// TwinCAT 3 PLC project Plc
// ProgramVersion: 3.1.4024.0
// libraries:
//   Tc2_Standard, * (Beckhoff Automation GmbH)
//   Tc2_System, * (Beckhoff Automation GmbH)
//   Tc3_Module, * (Beckhoff Automation GmbH)
//   VisuDialogs, * (System)
// project tree:
//   / Gestore di visualizzazione.TcVMO (not stored), GlobalTextList.TcGTLO, ImagePool.TcIPO (not stored), PlcTask.TcTTO (not stored), VisuTask.TcTTO
//   GVLs/ GVL.TcGVL
//   POUs/ MAIN.TcPOU, VISU.TcPOU (not stored)
//   VISUs/ Visualization.TcVIS
// real-time tasks:
//   TASK PlcTask: cycle T#10ms, priority 20, ADS port 350
//   TASK VisuTask: cycle T#100000us, priority 60, ADS port 351

CONFIGURATION Plc
    RESOURCE PLC ON TwinCAT3
        TASK VisuTask(INTERVAL := T#100000us, PRIORITY := 60);
        PROGRAM VISU WITH VisuTask : VISU;
    END_RESOURCE
END_CONFIGURATION

// ---- GVLs/GVL.TcGVL
{attribute 'qualified_only'}
VAR_GLOBAL
	//input
	PB1: BOOL; //Pulsante di start NA
	PB2: BOOL; //Pulsante di stop NC
	PBE: BOOL; //Pulsante di emergenza NC
	PS1: BOOL; //Fotocellula
	PS2: BOOL; //Fotocellula
	PS3: BOOL; //Fotocellula
	PS4: BOOL; //Fotocellula
	PS5: BOOL; //Fotocellula
	CS_BIANCO: BOOL; //Colore bianco rilevato
	CS_NERO: BOOL; //Colore nero rilevato
	
	//output
	L1: BOOL; //Luce di segnalazione bianca
	L2: BOOL; //Luce di segnalazione verde
	L3: BOOL; //Luce di segnalazione blue
	L4: BOOL; //Luce di segnalazione gialla
	L5: BOOL; //Luce di segnalazione rossa
	M1 : BOOL; //Motore nastro 1
	M2 : BOOL; //Motore nastro 2
	M3 : BOOL; //Motore discesa mandrino
	M4 : BOOL; //MOtore risalita mandrino
	M5 : BOOL; //Punta del trapano
	P1 : BOOL; //Pistone posizione intermedia
	P2 : BOOL; //Pistone posizione finale
	P3 : BOOL; //Pistone timbratura
	P4 : BOOL; //Pistone blocco pezzo
END_VAR

// ---- POUs/MAIN.TcPOU
PROGRAM MAIN
VAR
	//Stati
	IN_FUNZIONE: BOOL;
	IN_SMISTAMENTO: BOOL;
	IN_TIMBRATURA: BOOL;
	IN_FORATURA: BOOL;
	PEZZO_BIANCO: BOOL;
	PEZZO_NERO: BOOL;
	
	//Timer
	TON_BIANCO: TON;
	TON_NERO: TON;
	TON_TIMBRATURA: TON;
	TON_FORATURA_1: TON; // Il trapano scende in 2 secondi
	TON_FORATURA_2: TON; // Il trapano risale in 2 secondi

	//Counter
	CTU_BIANCHI: CTU;
	CTU_NERI: CTU;
	STOP_CONFERMATO: BOOL;
	STOP_RICHIESTO: BOOL;
	TON_STOP: TON;
	IN_ANOMALIA: BOOL;
	TON_ANOMALIA: TON;
	CONTROLLO_COLORE: BOOL;
	TON_ANOMALIA_COLORE: TON;
END_VAR

GestioneAnomalie();
GestioneStop();
GestionePulsantiSegnalazioni();
GestioneMotori();
GestioneSmistamento();
GestioneTimbratura();
GestioneForatura();
GestioneConteggio();

ACTION GestioneAnomalie:
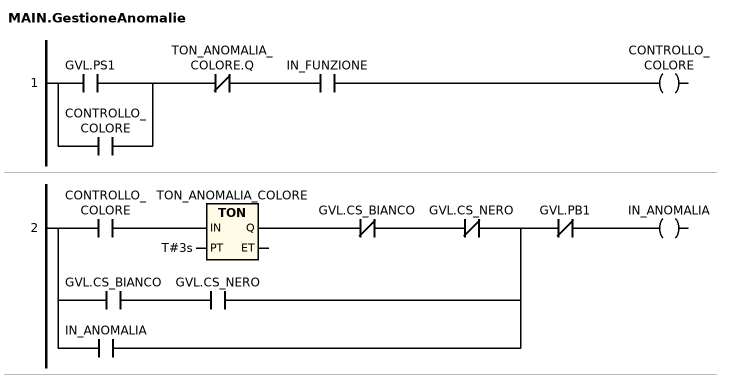
// NETWORK 1
CONTROLLO_COLORE := (GVL.PS1 OR CONTROLLO_COLORE) AND NOT TON_ANOMALIA_COLORE.Q AND IN_FUNZIONE;

// NETWORK 2
TON_ANOMALIA_COLORE(IN := CONTROLLO_COLORE, PT := T#3s); // TON
IN_ANOMALIA := (TON_ANOMALIA_COLORE.Q AND NOT GVL.CS_BIANCO AND NOT GVL.CS_NERO OR GVL.CS_BIANCO AND GVL.CS_NERO OR IN_ANOMALIA) AND NOT GVL.PB1;
END_ACTION

ACTION GestioneConteggio:
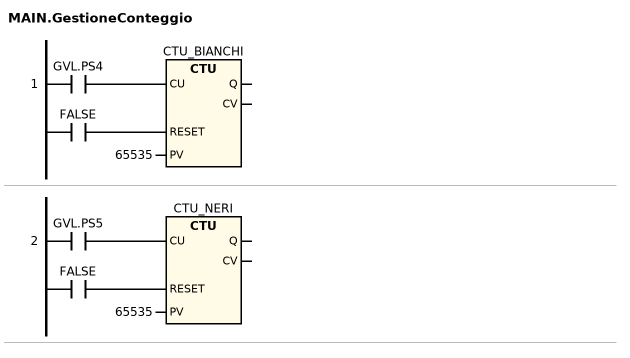
// NETWORK 1
CTU_BIANCHI(CU := GVL.PS4, RESET := FALSE, PV := 65535); // CTU

// NETWORK 2
CTU_NERI(CU := GVL.PS5, RESET := FALSE, PV := 65535); // CTU
END_ACTION

ACTION GestioneForatura:
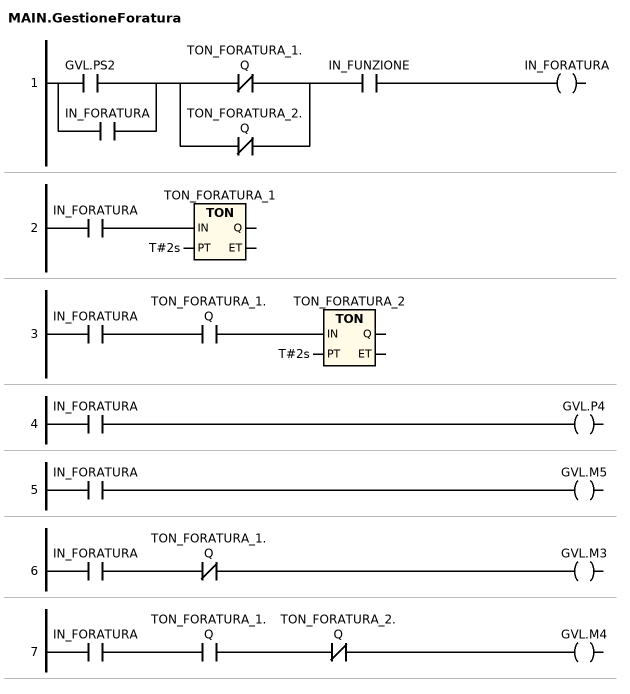
// NETWORK 1
IN_FORATURA := (GVL.PS2 OR IN_FORATURA) AND (NOT TON_FORATURA_1.Q OR NOT TON_FORATURA_2.Q) AND IN_FUNZIONE;

// NETWORK 2
TON_FORATURA_1(IN := IN_FORATURA, PT := T#2s); // TON

// NETWORK 3
TON_FORATURA_2(IN := IN_FORATURA AND TON_FORATURA_1.Q, PT := T#2s); // TON

// NETWORK 4
GVL.P4 := IN_FORATURA;

// NETWORK 5
GVL.M5 := IN_FORATURA;

// NETWORK 6
GVL.M3 := IN_FORATURA AND NOT TON_FORATURA_1.Q;

// NETWORK 7
GVL.M4 := IN_FORATURA AND TON_FORATURA_1.Q AND NOT TON_FORATURA_2.Q;
END_ACTION

ACTION GestioneMotori:
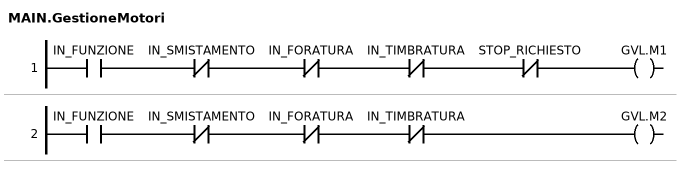
// NETWORK 1
GVL.M1 := IN_FUNZIONE AND NOT IN_SMISTAMENTO AND NOT IN_FORATURA AND NOT IN_TIMBRATURA AND NOT STOP_RICHIESTO;

// NETWORK 2
GVL.M2 := IN_FUNZIONE AND NOT IN_SMISTAMENTO AND NOT IN_FORATURA AND NOT IN_TIMBRATURA;
END_ACTION

ACTION GestionePulsantiSegnalazioni:
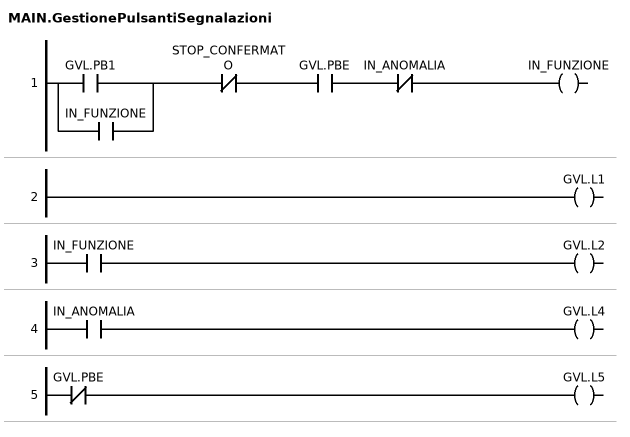
// NETWORK 1
IN_FUNZIONE := (GVL.PB1 OR IN_FUNZIONE) AND NOT STOP_CONFERMATO AND GVL.PBE AND NOT IN_ANOMALIA;

// NETWORK 2
GVL.L1 := TRUE;

// NETWORK 3
GVL.L2 := IN_FUNZIONE;

// NETWORK 4
GVL.L4 := IN_ANOMALIA;

// NETWORK 5
GVL.L5 := NOT GVL.PBE;
END_ACTION

ACTION GestioneSmistamento:
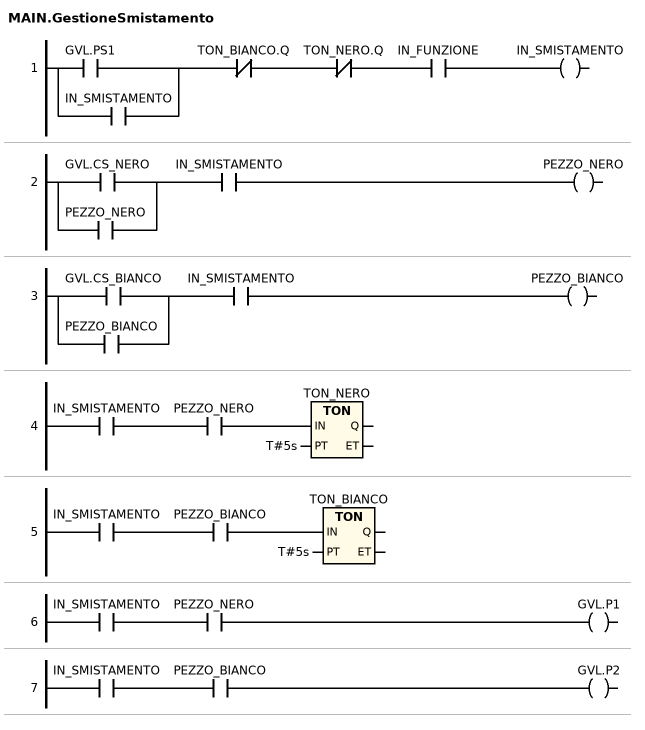
// NETWORK 1
IN_SMISTAMENTO := (GVL.PS1 OR IN_SMISTAMENTO) AND NOT TON_BIANCO.Q AND NOT TON_NERO.Q AND IN_FUNZIONE;

// NETWORK 2
PEZZO_NERO := (GVL.CS_NERO OR PEZZO_NERO) AND IN_SMISTAMENTO;

// NETWORK 3
PEZZO_BIANCO := (GVL.CS_BIANCO OR PEZZO_BIANCO) AND IN_SMISTAMENTO;

// NETWORK 4
TON_NERO(IN := IN_SMISTAMENTO AND PEZZO_NERO, PT := T#5s); // TON

// NETWORK 5
TON_BIANCO(IN := IN_SMISTAMENTO AND PEZZO_BIANCO, PT := T#5s); // TON

// NETWORK 6
GVL.P1 := IN_SMISTAMENTO AND PEZZO_NERO;

// NETWORK 7
GVL.P2 := IN_SMISTAMENTO AND PEZZO_BIANCO;
END_ACTION

ACTION GestioneStop:
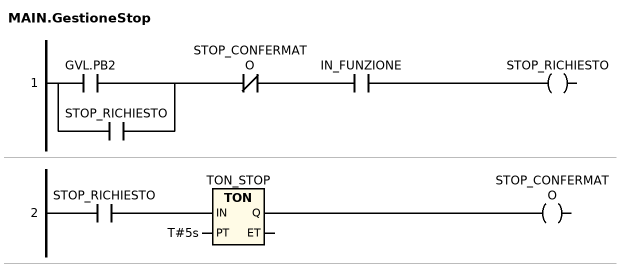
// NETWORK 1
STOP_RICHIESTO := (GVL.PB2 OR STOP_RICHIESTO) AND NOT STOP_CONFERMATO AND IN_FUNZIONE;

// NETWORK 2
TON_STOP(IN := STOP_RICHIESTO, PT := T#5s); // TON
STOP_CONFERMATO := TON_STOP.Q;
END_ACTION

ACTION GestioneTimbratura:
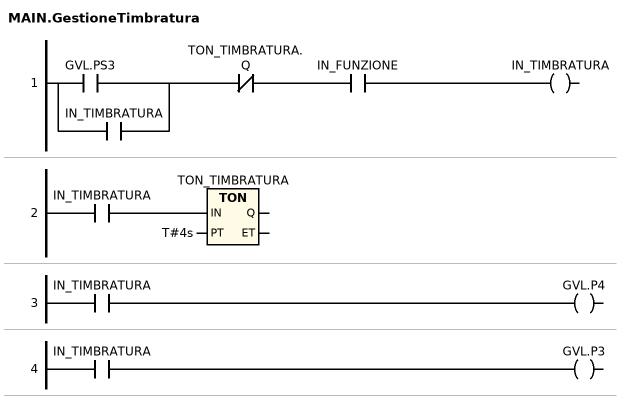
// NETWORK 1
IN_TIMBRATURA := (GVL.PS3 OR IN_TIMBRATURA) AND NOT TON_TIMBRATURA.Q AND IN_FUNZIONE;

// NETWORK 2
TON_TIMBRATURA(IN := IN_TIMBRATURA, PT := T#4s); // TON

// NETWORK 3
GVL.P4 := IN_TIMBRATURA;

// NETWORK 4
GVL.P3 := IN_TIMBRATURA;
END_ACTION

END_PROGRAM

// ---- GlobalTextList.TcGTLO
TEXTLIST GlobalTextList
  628 = '%d'
  216 = '%f'
  108 = 'A11'
  331 = 'A12'
  600 = 'B11'
  978 = 'C'
  333 = 'C11'
  372 = 'CS_BIANCO'
  547 = 'CS_NERO'
  68 = 'Emergenza'
  428 = 'EMERGENZA'
  304 = 'foratura'
  801 = 'FS1'
  524 = 'FS2'
  765 = 'LC1'
  869 = 'M1'
  802 = 'M2'
  115 = 'M3'
  287 = 'M4'
  498 = 'M5'
  501 = 'Percentuale prosciutti commerciabili: %d'
  820 = 'Percentuale prosciutti commerciabili:%d'
  57 = 'pistone'
  388 = 'PS1'
  310 = 'PS2'
  806 = 'PS3'
  525 = 'PS4'
  656 = 'SB1'
  665 = 'SB2'
  112 = 'SB3'
  871 = 'Start'
  375 = 'START'
  275 = 'Stop'
  437 = 'STOP'
  800 = 'timbratura'
  305 = 'vasca di contenimento '
END_TEXTLIST

// ---- VISUs/Visualization.TcVIS
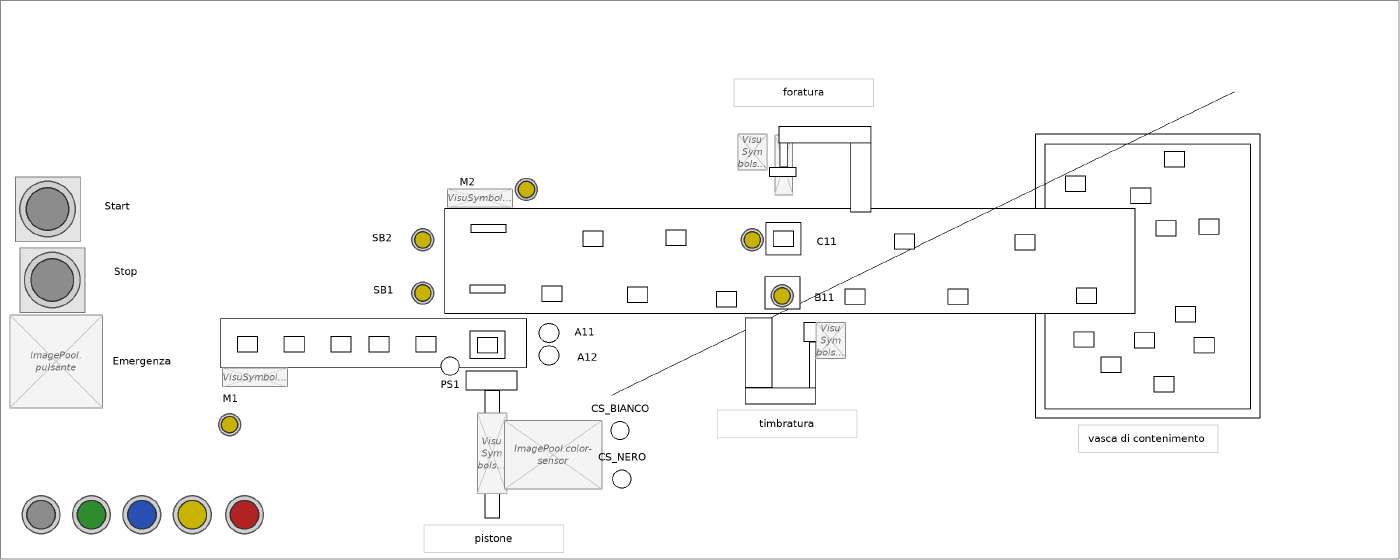
VISUALIZATION Visualization  // 1500x600
    PushSwitch (16,189 70x70), variable: GVL.PB1, behaviour: TAP, style: Switch-PushSwitch-Gray
    Label (98,206 55x30), "Start"
    PushSwitch (21,265 70x70), variable: GVL.PB2, behaviour: TAP, style: Switch-PushSwitch-Gray
    Label (102,276 65x30), "Stop"
    Label (107,372 90x30), "Emergenza"
    Lamp1 (20,527 48x49), variable: GVL.L1, style: Lamp-Lamp1-Gray
    Lamp1 (74,527 48x49), variable: GVL.L2, style: Lamp-Lamp1-Green
    Lamp1 (128,527 48x49), variable: GVL.L3, style: Lamp-Lamp1-Blue
    Lamp1 (182,527 48x49), variable: GVL.L4, style: Lamp-Lamp1-Yellow
    Lamp1 (238,527 48x49), variable: GVL.L5, style: Lamp-Lamp1-Red
    Image (10,337 100x100), image: ImagePool.pulsante
        OnMouseClick: toggle GVL.PBE
    Textfield (454,562 150x30), "pistone"
    Image (830,144 19x65), image: VisuSymbols.Symbols.ArrowBoldDown
    RoundedRectangle (1109,143 241x305)
    RoundedRectangle (1119,154 221x284)
    Rectangle (236,341 328x53)
    RoundedRectangle (476,223 740x113)
    Line (655,423) (1322,98)
    RoundedRectangle (499,397 55x21)
    Rectangle (519,418 16x137)
    Image (511,442 32x87), image: VisuSymbols.Symbols.DoubleArrow4
    Rectangle (254,360 22x17)
    Rectangle (304,360 22x17)
    Rectangle (354,360 22x17)
    Rectangle (395,360 22x17)
    Rectangle (624,247 22x17)
    Rectangle (713,246 22x17)
    Rectangle (445,360 22x17)
    Rectangle (580,306 22x17)
    Rectangle (672,307 22x17)
    Rectangle (767,312 22x17)
    Rectangle (905,309 22x17)
    Rectangle (1015,309 22x17)
    Rectangle (1153,308 22x17)
    Rectangle (958,250 22x17)
    Rectangle (1087,251 22x17)
    Rectangle (1179,382 22x17)
    Rectangle (1279,361 22x17)
    Rectangle (1259,328 22x17)
    Rectangle (1215,356 22x17)
    Rectangle (1150,355 22x17)
    Rectangle (1236,403 22x17)
    Rectangle (1141,188 22x17)
    Rectangle (1211,201 22x17)
    Rectangle (1247,162 22x17)
    Rectangle (1238,236 22x17)
    Rectangle (1284,234 22x17)
    Textfield (1155,455 150x30), "vasca di contenimento"
    RoundedRectangle (861,345 19x21)
    Rectangle (867,366 7x51)
    Rectangle (798,415 76x18)
    Rectangle (798,340 29x75)
    Image (874,345 32x39), image: VisuSymbols.Symbols.DoubleArrow4
    Textfield (768,439 150x30), "timbratura"
    Textfield (786,84 150x30), "foratura"
    Rectangle (911,152 22x75)
    RoundedRectangle (824,179 29x10)
    Rectangle (835,150 9x29)
    Rectangle (834,135 99x18)
    Image (790,143 32x39), image: VisuSymbols.Symbols.DoubleArrow4
    Image (479,202 70x20), image: VisuSymbols.Symbols.ArrowBoldRight
    Image (238,394 70x20), image: VisuSymbols.Symbols.ArrowBoldRight
    Rectangle (503,354 38x30)
    Rectangle (511,361 22x17)
    Rectangle (820,238 38x35)
    Rectangle (819,296 38x35)
    Rectangle (828,247 22x17)
    Rectangle (504,240 38x9)
    Rectangle (503,305 38x9)
    Lamp1 (439,242 28x30), variable: MAIN.SB2, style: Lamp-Lamp1-Yellow
    Lamp1 (439,299 28x30), variable: MAIN.SB1, style: Lamp-Lamp1-Yellow
    Lamp1 (824,302 28x30), variable: MAIN.B1, style: Lamp-Lamp1-Yellow
    Lamp1 (792,242 28x30), variable: MAIN.C1, style: Lamp-Lamp1-Yellow
    Label (205,412 84x30), "M1"
    Label (459,180 84x30), "M2"
    Label (600,341 53x30), "A11"
    Label (858,244 56x30), "C11"
    Label (605,368 49x30), "A12"
    Label (388,296 46x30), "SB1"
    Label (385,240 49x30), "SB2"
    Label (855,304 57x30), "B11"
    Ellipse (577,346 22x21)
        tap MAIN.A11
    Ellipse (577,370 22x21)
        tap MAIN.A12
    Lamp1 (232,440 28x30), variable: MAIN.motore1, style: Lamp-Lamp1-Yellow
    Lamp1 (550,188 28x30), variable: MAIN.motore2, style: Lamp-Lamp1-Yellow
    Ellipse (654,451 20x20), colour toggle: GVL.M1
    Label (622,432 85x12), "CS_BIANCO"
    Ellipse (472,382 20x20), colour toggle: GVL.M1
    Label (463,406 39x12), "PS1"
    Image (540,450 105x74), image: ImagePool.color-sensor
    Ellipse (656,503 20x20), colour toggle: GVL.M1
    Label (624,484 85x12), "CS_NERO"
END_VISUALIZATION
